{attribute 'qualified_only'}
VAR_GLOBAL
	station:typeStation; //data relating to the entire station
END_VAR

(* stored: Version 1.1.0.1, ProductVersion 3.1.4024.12
   GVL S3_Global: Id {82adc27a-2641-4265-86c8-415bf9768a73} *)
